(*

.. <legal notes>

legal notes
=================
| SPDX-FileCopyrightText: © 2026 Oleksandr Tiutyk <trofimich@gmail.com>
| SPDX-License-Identifier: LGPL-3.0-only
| For details check: LGPL-3.0-only_

.. _LGPL-3.0-only: https://www.gnu.org/licenses/lgpl-3.0.en.html

.. </legal notes>

*)

{attribute 'no_explicit_call' := 'do not call this POU directly'}
PROGRAM CurrentNamespace
VAR
	_NamespaceExtractor : NamespaceExtractor;
END_VAR

{attribute 'monitoring' := 'call'}
PROPERTY Name : STRING
GET
Name := _NamespaceExtractor.CurrentNamespace;
END_GET
END_PROPERTY

END_PROGRAM

(* stored: Version 1.1.0.1
   POU CurrentNamespace: Id {4340c815-7bca-4048-a45a-a862e4b07ee7}, SpecialFunc None
   Property Name: Id {2eedbc7c-0c57-4efb-be33-1f26bf160a8f}
   Get Get: Id {1c8f1056-21b1-4feb-9761-1f223891c41c} *)
